//{attribute 'qualified_only'}
//{attribute 'strict'}
{attribute 'to_string'}
{attribute 'to_wstring'}
TYPE E_St050_Settings :
(
	//eSt050_Settings_none := 0,
	
	eSt050_Settings_Station_Deaktiv,	// Station deaktivieren
	eSt050_Settings_Autohome,			// automatic home with start button

	
	/// has to be set to last index for array bounds!
	eSt050_Settings_nMaxIdx	
);
END_TYPE

(* stored: Version 1.1.0.1
   DUT E_St050_Settings: Id {ee1341f6-d38a-4579-bd85-e028817b4b74} *)
